(* CODESYS project PLC_PRG.export

Project tree, tasks and I/O mapping:
  program PLC_PRG [ST]
*)

// PLC_PRG
PROGRAM PLC_PRG
VAR 
	(**** SENSOR EDGES ****)
	F_AtEntry           : F_TRIG;
    F_AtTurnEntry       : F_TRIG;
    F_AtRightEntry      : F_TRIG;
    F_AtLeftEntry       : F_TRIG;
    F_AtRightExit       : F_TRIG;
    F_AtLeftExit        : F_TRIG;
	(**** LEFT EXIT CONVEYER STATES ****)
    Pallet_on_left      : BOOL := FALSE;
	(**** RIGHT EXIT CONVEYER STATES ****)
    Pallet_on_right     : BOOL := FALSE;
	(**** TURNTABLE STATES ****)
    Idle                : BOOL := TRUE;
    Charging            : BOOL := FALSE;
    Turns_charged       : BOOL := FALSE;
    Discharging         : BOOL := FALSE;
    Turns_Discharged    : BOOL := FALSE;
    Turntable_busy      : BOOL := FALSE;
    Discharge_direction : BOOL := FALSE;
	Discharge_direction_temp : BOOL := FALSE;
	HeightTimer			:TON;
	(**** ENTRY CONVEYER STATES ****)
    Entry_busy          : BOOL := FALSE;
    Pallet_on_entry     : BOOL := FALSE;
    CountLeft               : INT := 0;
	CountRight               : INT := 0;
END_VAR

(**** FLASHER ****)
GVL.blinker(IN:= NOT GVL.blinker.Q,PT :=T#1000MS);
IF GVL.blinker.ET <= T#500MS THEN
	GVL.flash := TRUE;
ELSE GVL.flash := FALSE;
END_IF

(**** OPERATION MODES ****)

GVL.Auto := FIO.iAuto AND NOT FIO.iManual;
GVL.Manual := FIO.iManual AND NOT FIO.iAuto;

IF GVL.Auto AND FIO.iStart AND NOT GVL.E_Stop AND NOT GVL.Confirmation_Required THEN
	GVL.Auto_Run := TRUE;
	GVL.Auto_Stop := FALSE;
ELSIF (GVL.Auto AND GVL.Auto_Run AND NOT FIO.iStop) THEN 
	GVL.Auto_Run := FALSE;
	GVL.Auto_Stop := TRUE;
END_IF;

IF GVL.E_Stop OR GVL.Confirmation_Required OR GVL.Manual THEN
	GVL.Auto_Run := FALSE;
	GVL.Auto_Stop := FALSE;
END_IF;

FIO.oStartLight := GVL.Auto_Run OR (GVL.Auto AND NOT GVL.Auto_Run AND NOT GVL.Auto_Stop AND NOT GVL.E_Stop AND NOT GVL.Confirmation_Required AND GVL.flash);
FIO.oStopLight := GVL.Auto_Stop;

(**** Skip all states in manual with RESET****)
IF GVL.Manual AND FIO.iReset THEN
	Pallet_on_left 		:= FALSE;
	Pallet_on_right 	:= FALSE;
	Idle                := TRUE;
    Charging            := FALSE;
    Turns_charged       := FALSE;
    Discharging         := FALSE;
    Turns_Discharged    := FALSE;
    Turntable_busy      := FALSE;
    Discharge_direction := FALSE;
	Entry_busy          := FALSE;
    Pallet_on_entry     := FALSE;
    CountLeft           := 0;
	CountRight          := 0;
END_IF

(**** E-STOP ****)
GVL.E_Stop := NOT FIO.iEmergencyStop;
IF NOT FIO.iEmergencyStop THEN
	GVL.Confirmation_Required := TRUE;
END_IF
FIO.oResetLight := GVL.Confirmation_Required AND GVL.flash;
IF GVL.Confirmation_Required AND FIO.iReset AND NOT GVL.E_Stop THEN
	GVL.Confirmation_Required := FALSE;
END_IF

(**** SENSOR EDGES ****)
F_AtEntry(CLK := FIO.iAtEntry);
F_AtTurnEntry(CLK := FIO.iAtTurnEntry);
F_AtRightEntry(CLK := FIO.iAtRightEntry);
F_AtLeftEntry(CLK := FIO.iAtLeftEntry);     (* A pallet abandons the turntable, being charged onto the left exit conveyer *)
F_AtRightExit(CLK := FIO.iAtRightExit);
F_AtLeftExit(CLK := FIO.iAtLeftExit);       (* A pallet abandons the left exit conveyer *)

(**** LEFT EXIT CONVEYER CONTROL ****)
(* Pallet_on_left represents the state of the left exit conveyer: if it carries a pallet, then Pallet_on_left = TRUE *)

IF F_AtLeftExit.Q THEN                      (* When a pallet abandons the conveyer *)
    Pallet_on_left := FALSE;                (* Reset Pallet_on_left *)
END_IF;

IF FIO.iAtLeftEntry THEN                    (* When there’s a pallet at the entry of the conveyer *)
    Pallet_on_left := TRUE;                 (* Set Pallet_on_left *)
END_IF;

FIO.oLeftConveyor := (Pallet_on_left AND GVL.Auto_Run) OR 
(GVL.Manual AND FIO.buttonLeftConveyor AND NOT GVL.E_Stop AND NOT GVL.Confirmation_Required);        (* Left exit conveyer runs for Pallet_on_left = TRUE *)

(**** RIGHT EXIT CONVEYER CONTROL ****)

IF F_AtRightExit.Q THEN
    Pallet_on_right := FALSE;
END_IF;

IF FIO.iAtRightEntry THEN
    Pallet_on_right := TRUE;
END_IF;

FIO.oRightConveyor := (Pallet_on_right AND GVL.Auto_Run) OR 
(GVL.Manual AND FIO.buttonRightConveyor AND NOT GVL.E_Stop AND NOT GVL.Confirmation_Required);

(**** TURNTABLE CONTROL ****)

IF Idle AND FIO.iAtTurnEntry THEN
    Idle := FALSE;
    Charging := TRUE;
END_IF;

IF Charging AND FIO.iAtFront THEN
    Charging := FALSE;
    Turns_charged := TRUE;
END_IF;

IF Turns_charged AND FIO.iAtUnloadPos THEN
    Turns_charged := FALSE;
    Discharging := TRUE;
END_IF;

(* The turntable discharges now onto both conveyers. Thus: *)

IF Discharging AND (F_AtRightEntry.Q OR F_AtLeftEntry.Q) THEN
    Discharging := FALSE;
    Turns_Discharged := TRUE;
END_IF;

IF Turns_Discharged AND FIO.iAtLoadPos THEN
    Turns_Discharged := FALSE;
    Idle := TRUE;
END_IF;

IF F_AtTurnEntry.Q THEN
    Turntable_busy := TRUE;
END_IF;

IF Idle THEN
    Turntable_busy := FALSE;
END_IF;

(* Computing control outputs according to the current state of the turntable and the direction of the discharge *)
FIO.oLoad := ((Charging OR Discharging AND Discharge_direction) AND GVL.Auto_Run) OR 
(GVL.Manual AND FIO.buttonLoad AND NOT GVL.E_Stop AND NOT GVL.Confirmation_Required);

(* oUnload is TRUE if the discharge is onto the left conveyer *)
FIO.oUnload := ((Discharging AND NOT Discharge_direction) AND GVL.Auto_Run) OR 
(GVL.Manual AND FIO.buttonUnload AND NOT GVL.E_Stop AND NOT GVL.Confirmation_Required);

(* oTurn is TRUE if the discharge is onto the right conveyer *)
FIO.oTurn := ((Turns_charged OR Discharging) AND GVL.Auto_Run) OR 
(GVL.Manual AND FIO.buttonTurn AND NOT GVL.E_Stop AND NOT GVL.Confirmation_Required);

(**** ENTRY CONVEYER CONTROL ****)
IF F_AtEntry.Q THEN
        Entry_busy := TRUE;
END_IF;

HeightTimer(IN:=FIO.iLowBox,PT:=T#500ms);
IF FIO.iLowBox AND NOT FIO.iHighBox AND HeightTimer.Q THEN
	Discharge_direction_temp := FALSE;
END_IF;
IF FIO.iLowBox AND  FIO.iHighBox AND HeightTimer.Q THEN
	Discharge_direction_temp := TRUE;
END_IF;

IF F_AtTurnEntry.Q THEN
(** Defining the direction of the discharge: the direction of the discharge changes every time a pallet is
discharged from the entry conveyer onto the turntable. If Discharge_direction = FALSE, then the discharge is onto the right conveyer **)
    Entry_busy := FALSE;
    Pallet_on_entry := FALSE;
	Discharge_direction:=Discharge_direction_temp;
END_IF;

IF FIO.iAtEntry THEN
    Pallet_on_entry := TRUE;
END_IF;

FIO.oEntryConveyor := (Pallet_on_entry AND (NOT Turntable_busy OR NOT FIO.iAtTurnEntry) AND GVL.Auto_Run) OR (GVL.Manual AND FIO.buttonEntryConveyor AND NOT GVL.E_Stop AND NOT GVL.Confirmation_Required);

(**** FEEDING CONVEYER CONTROL ****)
FIO.oFeederConveyor := ((NOT Entry_busy OR NOT FIO.iAtEntry) AND GVL.Auto_Run) OR 
(GVL.Manual AND FIO.buttonFeederConveyor AND NOT GVL.E_Stop AND NOT GVL.Confirmation_Required);

(**** COUNTER LEFT SIDE****)
IF F_AtLeftExit.Q  THEN
	CountLeft := CountLeft + 1;
END_IF
IF F_AtRightExit.Q  THEN
	CountRight := CountRight + 1;
END_IF

FIO.ointCounter := CountLeft + CountRight;

END_PROGRAM
